FUNCTION_BLOCK FB_HMIVision EXTENDS FB_HMIBase
VAR
	vision : Vision.I_Vision;  // Using interface for polymorphism
END_VAR

METHOD Cyclic
VAR
END_VAR
// Sync status from vision to HMI
IF __ISVALIDREF(vision.P_BaseStatus) THEN
	status.HmiStatus.Busy := vision.P_BaseStatus.Busy;
	status.HmiStatus.Error := vision.P_BaseStatus.Error;
	status.HmiStatus.ErrorID := UDINT_TO_BYTE(vision.P_BaseStatus.ErrorID);
END_IF

// Use handshake status for Done flag
IF __ISVALIDREF(vision.P_HandshakeStatus) THEN
	status.HmiStatus.Done := vision.P_HandshakeStatus.ResultsReceived;
END_IF

// Handle commands from Vue.js
IF cmd.Trigger THEN
	vision.Trigger();
	cmd.Trigger := FALSE;
END_IF
END_METHOD

METHOD FB_init : BOOL
VAR_INPUT
	bInitRetains : BOOL; // if TRUE, the retain variables are initialized (warm start / cold start)
	bInCopyCode : BOOL;  // if TRUE, the instance afterwards gets moved into the copy code (online change)
END_VAR
// Standard FB constructor - no custom initialization needed
END_METHOD

METHOD Init : BOOL
VAR_INPUT
	refVision : Vision.I_Vision;
END_VAR
vision := refVision;
Init := TRUE;
END_METHOD

END_FUNCTION_BLOCK

(* stored: Version 1.1.0.1
   POU FB_HMIVision: Id {b76f3680-5def-4f09-9741-0aa6629d1724}, SpecialFunc None
   Method Cyclic: Id {b43f8de0-78fb-4076-b614-792224a68729}
   Method FB_init: Id {8bbbca94-fa6c-4c61-9d57-8f6dfd6db76f}
   Method Init: Id {8bbbca95-fa6c-4c61-9d57-8f6dfd6db76f} *)
